(* Logix 5000 project; controller STAT 1756-L72 rev 20.12; software revision 20.04; part 7 of 34 *)
(* tags used below, declared in another part *)
   B11 : DINT[5];
   B15 : DINT[11];
   B3 : DINT[5];
   B9 : DINT[2];
   C5 : COUNTER[8];
   N17 : DINT[80];
   T10 : TIMER[30];
   T12 : TIMER[30];
   T4 : TIMER[30];
(* ECOTECH, continued *)

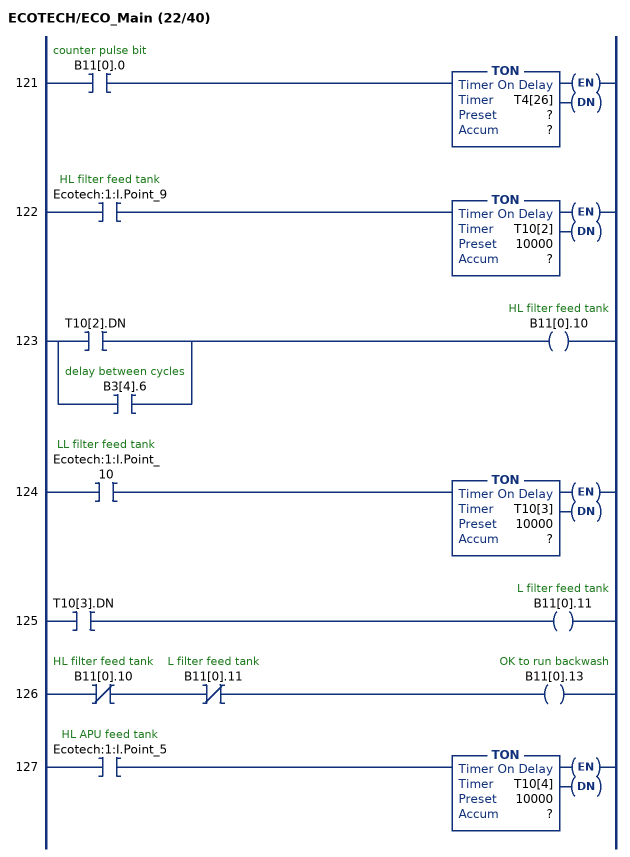
   [picture p70: ECOTECH/ECO_Main rungs 121-127]
   121: XIC(B11[0].0)TON(T4[26],?,?);
   122: XIC(Ecotech:1:I.Point_9)TON(T10[2],?,?);
   123: [XIC(T10[2].DN) ,XIC(B3[4].6) ]OTE(B11[0].10);
   124: XIC(Ecotech:1:I.Point_10)TON(T10[3],?,?);
   125: XIC(T10[3].DN)OTE(B11[0].11);
   126: XIO(B11[0].10)XIO(B11[0].11)OTE(B11[0].13);
   127: XIC(Ecotech:1:I.Point_5)TON(T10[4],?,?);
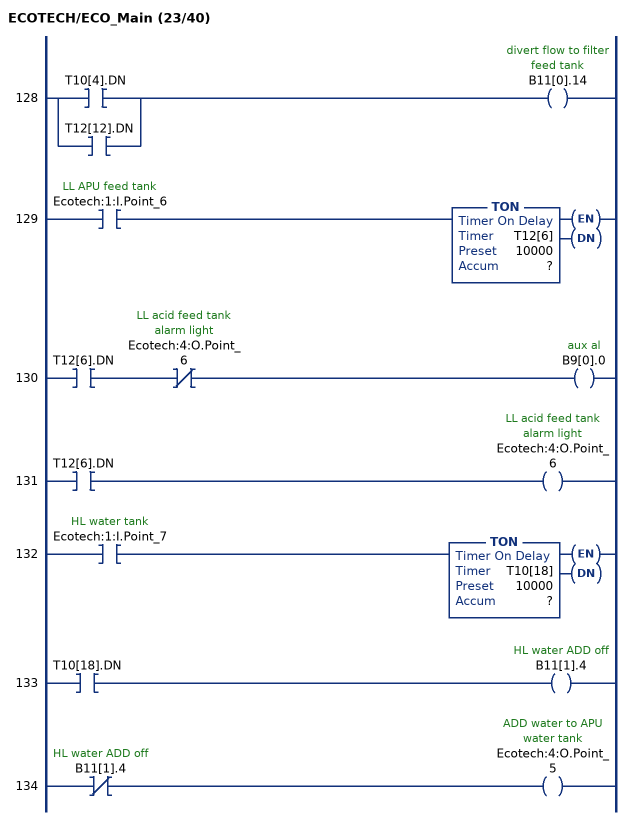
   128: [XIC(T10[4].DN) ,XIC(T12[12].DN) ]OTE(B11[0].14);
   129: XIC(Ecotech:1:I.Point_6)TON(T12[6],?,?);
   130: XIC(T12[6].DN)XIO(Ecotech:4:O.Point_6)OTE(B9[0].0);
   131: XIC(T12[6].DN)OTE(Ecotech:4:O.Point_6);
   132: XIC(Ecotech:1:I.Point_7)TON(T10[18],?,?);
   133: XIC(T10[18].DN)OTE(B11[1].4);
   134: XIO(B11[1].4)OTE(Ecotech:4:O.Point_5);
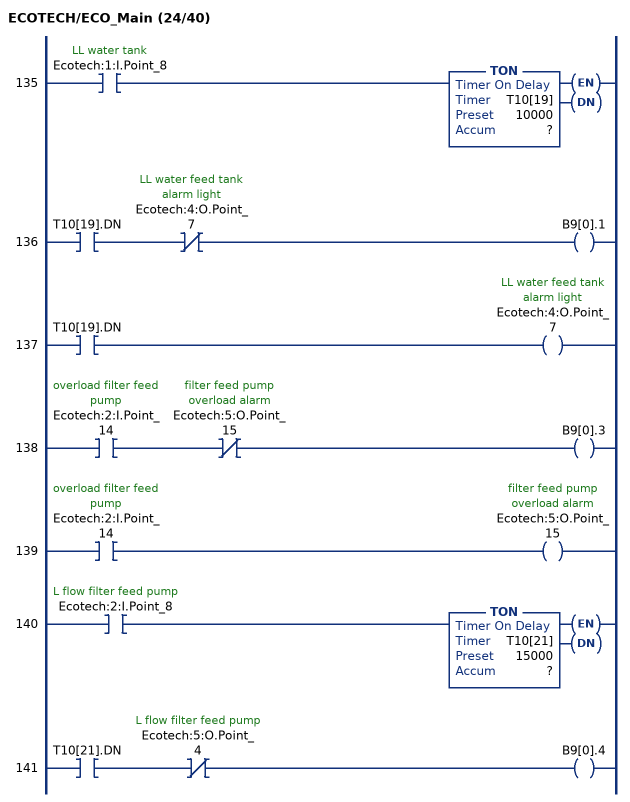
   135: XIC(Ecotech:1:I.Point_8)TON(T10[19],?,?);
   136: XIC(T10[19].DN)XIO(Ecotech:4:O.Point_7)OTE(B9[0].1);
   137: XIC(T10[19].DN)OTE(Ecotech:4:O.Point_7);
   138: XIC(Ecotech:2:I.Point_14)XIO(Ecotech:5:O.Point_15)OTE(B9[0].3);
   139: XIC(Ecotech:2:I.Point_14)OTE(Ecotech:5:O.Point_15);
   140: XIC(Ecotech:2:I.Point_8)TON(T10[21],?,?);
   141: XIC(T10[21].DN)XIO(Ecotech:5:O.Point_4)OTE(B9[0].4);
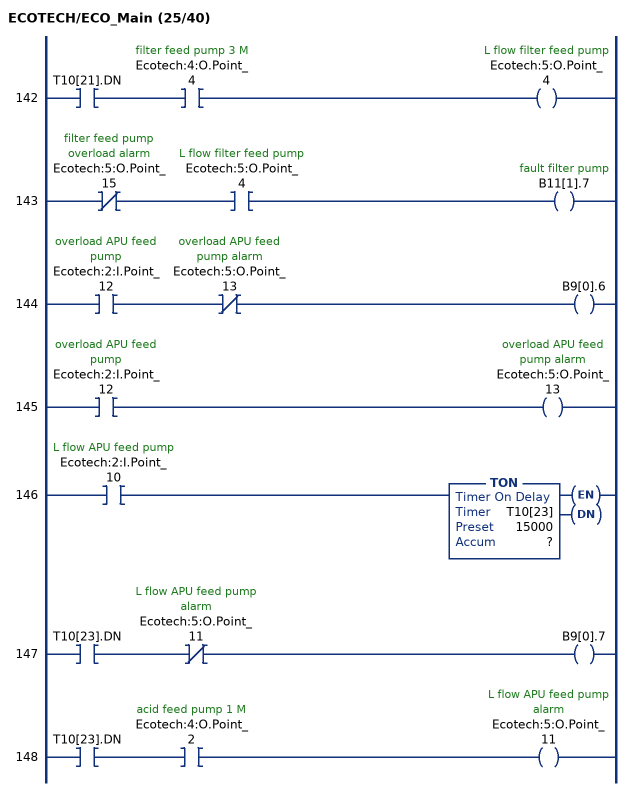
   142: XIC(T10[21].DN)XIC(Ecotech:4:O.Point_4)OTE(Ecotech:5:O.Point_4);
   143: XIO(Ecotech:5:O.Point_15)XIC(Ecotech:5:O.Point_4)OTE(B11[1].7);
   144: XIC(Ecotech:2:I.Point_12)XIO(Ecotech:5:O.Point_13)OTE(B9[0].6);
   145: XIC(Ecotech:2:I.Point_12)OTE(Ecotech:5:O.Point_13);
   146: XIC(Ecotech:2:I.Point_10)TON(T10[23],?,?);
   147: XIC(T10[23].DN)XIO(Ecotech:5:O.Point_11)OTE(B9[0].7);
   148: XIC(T10[23].DN)XIC(Ecotech:4:O.Point_2)OTE(Ecotech:5:O.Point_11);
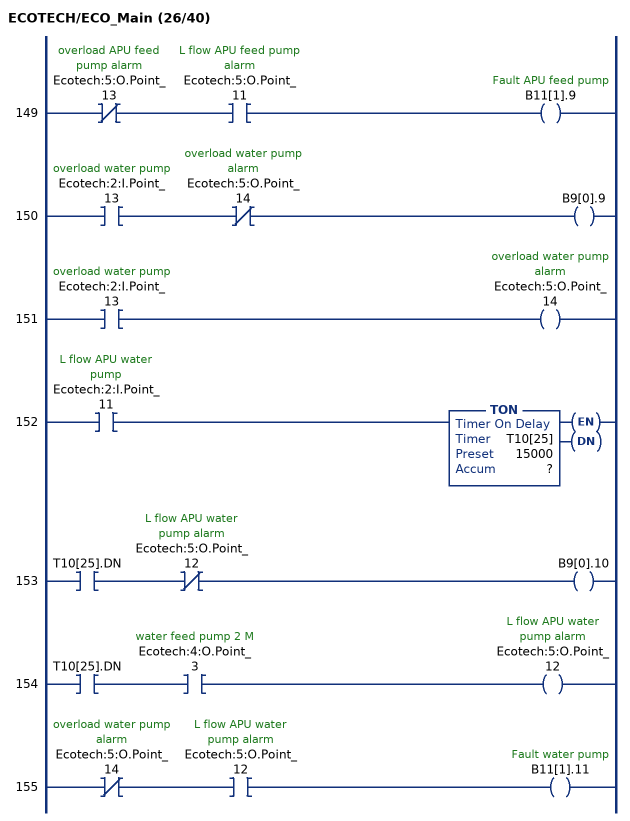
   149: XIO(Ecotech:5:O.Point_13)XIC(Ecotech:5:O.Point_11)OTE(B11[1].9);
   150: XIC(Ecotech:2:I.Point_13)XIO(Ecotech:5:O.Point_14)OTE(B9[0].9);
   151: XIC(Ecotech:2:I.Point_13)OTE(Ecotech:5:O.Point_14);
   152: XIC(Ecotech:2:I.Point_11)TON(T10[25],?,?);
   153: XIC(T10[25].DN)XIO(Ecotech:5:O.Point_12)OTE(B9[0].10);
   154: XIC(T10[25].DN)XIC(Ecotech:4:O.Point_3)OTE(Ecotech:5:O.Point_12);
   155: XIO(Ecotech:5:O.Point_14)XIC(Ecotech:5:O.Point_12)OTE(B11[1].11);
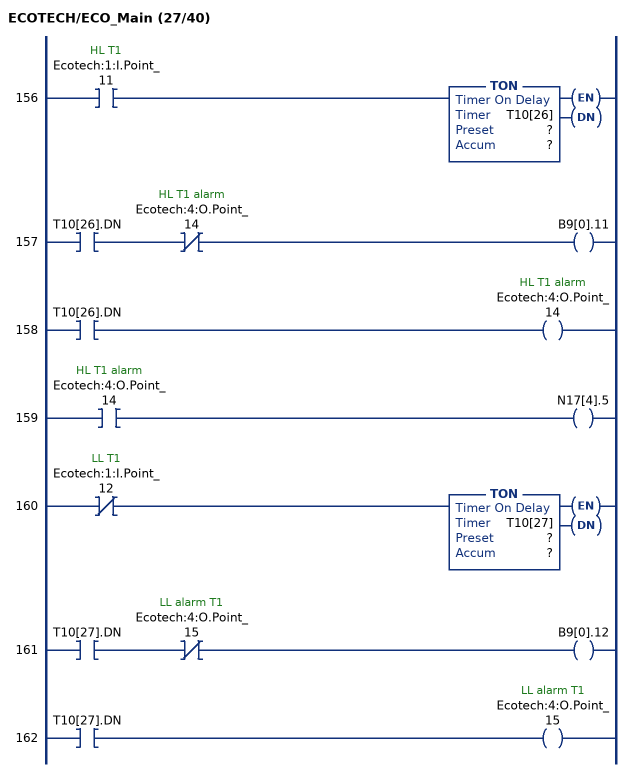
   156: XIC(Ecotech:1:I.Point_11)TON(T10[26],?,?);
   157: XIC(T10[26].DN)XIO(Ecotech:4:O.Point_14)OTE(B9[0].11);
   158: XIC(T10[26].DN)OTE(Ecotech:4:O.Point_14);
   159: XIC(Ecotech:4:O.Point_14)OTE(N17[4].5);
   160: XIO(Ecotech:1:I.Point_12)TON(T10[27],?,?);
   161: XIC(T10[27].DN)XIO(Ecotech:4:O.Point_15)OTE(B9[0].12);
   162: XIC(T10[27].DN)OTE(Ecotech:4:O.Point_15);
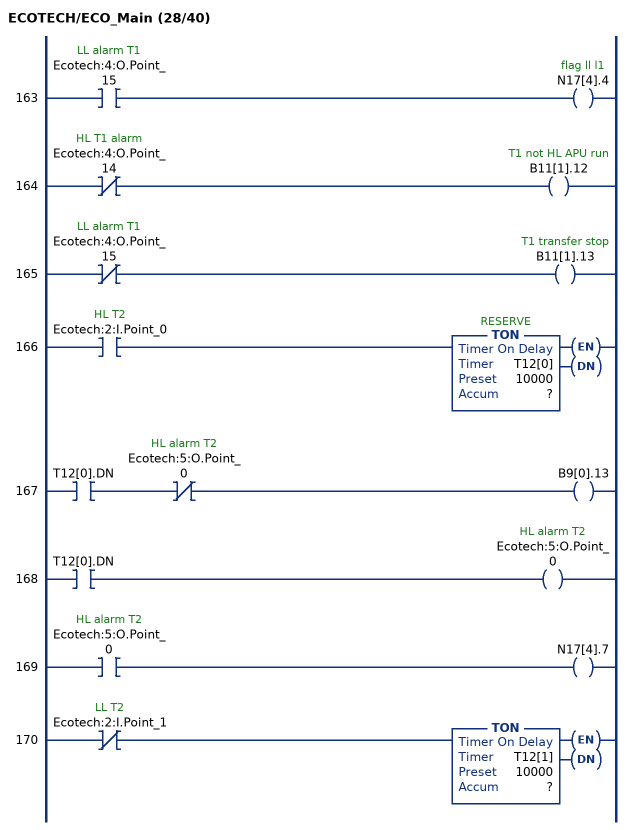
   163: XIC(Ecotech:4:O.Point_15)OTE(N17[4].4);
   164: XIO(Ecotech:4:O.Point_14)OTE(B11[1].12);
   165: XIO(Ecotech:4:O.Point_15)OTE(B11[1].13);
   166: XIC(Ecotech:2:I.Point_0)TON(T12[0],?,?);
   167: XIC(T12[0].DN)XIO(Ecotech:5:O.Point_0)OTE(B9[0].13);
   168: XIC(T12[0].DN)OTE(Ecotech:5:O.Point_0);
   169: XIC(Ecotech:5:O.Point_0)OTE(N17[4].7);
   170: XIO(Ecotech:2:I.Point_1)TON(T12[1],?,?);
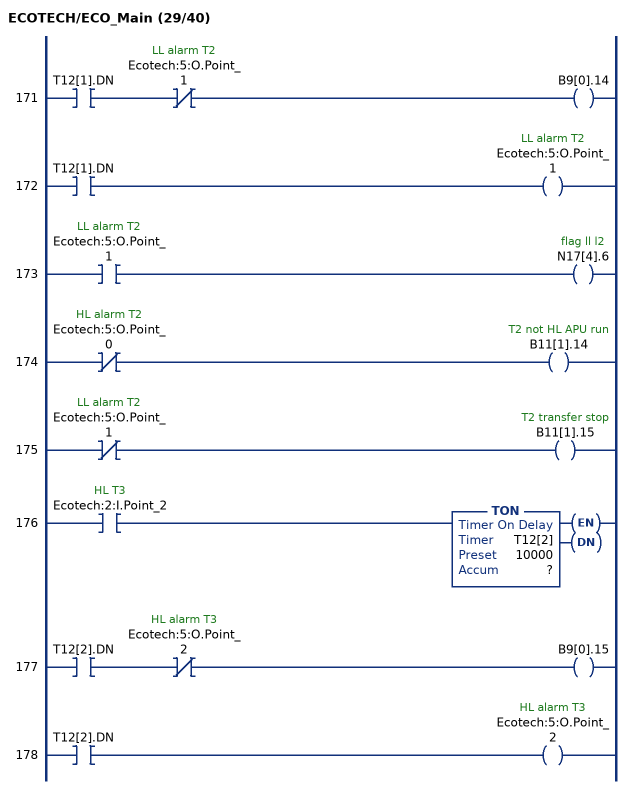
   171: XIC(T12[1].DN)XIO(Ecotech:5:O.Point_1)OTE(B9[0].14);
   172: XIC(T12[1].DN)OTE(Ecotech:5:O.Point_1);
   173: XIC(Ecotech:5:O.Point_1)OTE(N17[4].6);
   174: XIO(Ecotech:5:O.Point_0)OTE(B11[1].14);
   175: XIO(Ecotech:5:O.Point_1)OTE(B11[1].15);
   176: XIC(Ecotech:2:I.Point_2)TON(T12[2],?,?);
   177: XIC(T12[2].DN)XIO(Ecotech:5:O.Point_2)OTE(B9[0].15);
   178: XIC(T12[2].DN)OTE(Ecotech:5:O.Point_2);
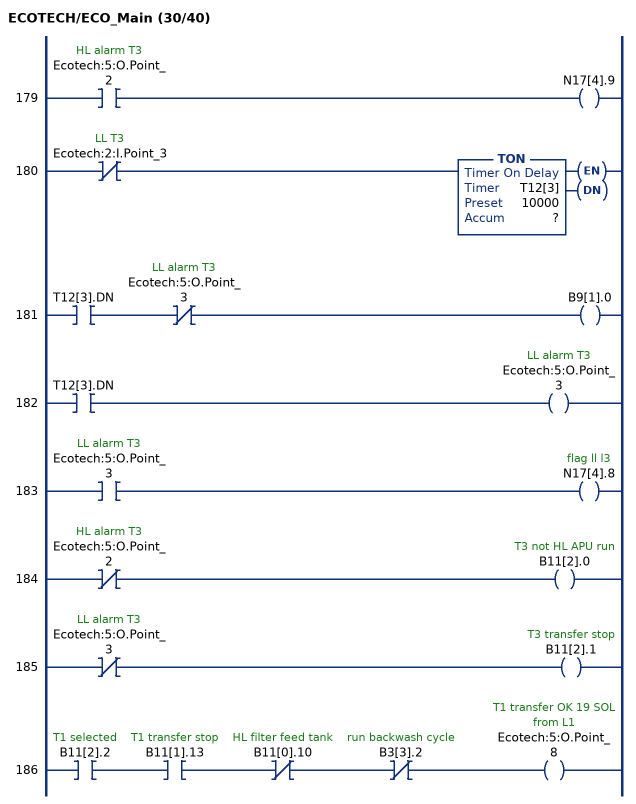
   179: XIC(Ecotech:5:O.Point_2)OTE(N17[4].9);
   180: XIO(Ecotech:2:I.Point_3)TON(T12[3],?,?);
   181: XIC(T12[3].DN)XIO(Ecotech:5:O.Point_3)OTE(B9[1].0);
   182: XIC(T12[3].DN)OTE(Ecotech:5:O.Point_3);
   183: XIC(Ecotech:5:O.Point_3)OTE(N17[4].8);
   184: XIO(Ecotech:5:O.Point_2)OTE(B11[2].0);
   185: XIO(Ecotech:5:O.Point_3)OTE(B11[2].1);
   186: XIC(B11[2].2)XIC(B11[1].13)XIO(B11[0].10)XIO(B3[3].2)OTE(Ecotech:5:O.Point_8);
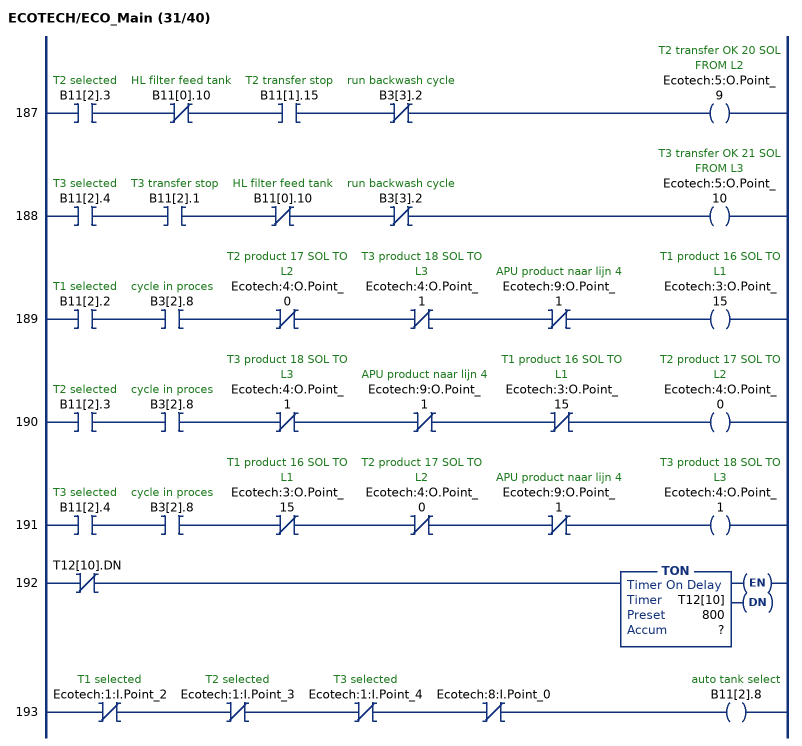
   187: XIC(B11[2].3)XIO(B11[0].10)XIC(B11[1].15)XIO(B3[3].2)OTE(Ecotech:5:O.Point_9);
   188: XIC(B11[2].4)XIC(B11[2].1)XIO(B11[0].10)XIO(B3[3].2)OTE(Ecotech:5:O.Point_10);
   189: XIC(B11[2].2)XIC(B3[2].8)XIO(Ecotech:4:O.Point_0)XIO(Ecotech:4:O.Point_1)XIO(Ecotech:9:O.Point_1)OTE(Ecotech:3:O.Point_15);
   190: XIC(B11[2].3)XIC(B3[2].8)XIO(Ecotech:4:O.Point_1)XIO(Ecotech:9:O.Point_1)XIO(Ecotech:3:O.Point_15)OTE(Ecotech:4:O.Point_0);
   191: XIC(B11[2].4)XIC(B3[2].8)XIO(Ecotech:3:O.Point_15)XIO(Ecotech:4:O.Point_0)XIO(Ecotech:9:O.Point_1)OTE(Ecotech:4:O.Point_1);
   192: XIO(T12[10].DN)TON(T12[10],?,?);
   193: XIO(Ecotech:1:I.Point_2)XIO(Ecotech:1:I.Point_3)XIO(Ecotech:1:I.Point_4)XIO(Ecotech:8:I.Point_0)OTE(B11[2].8);
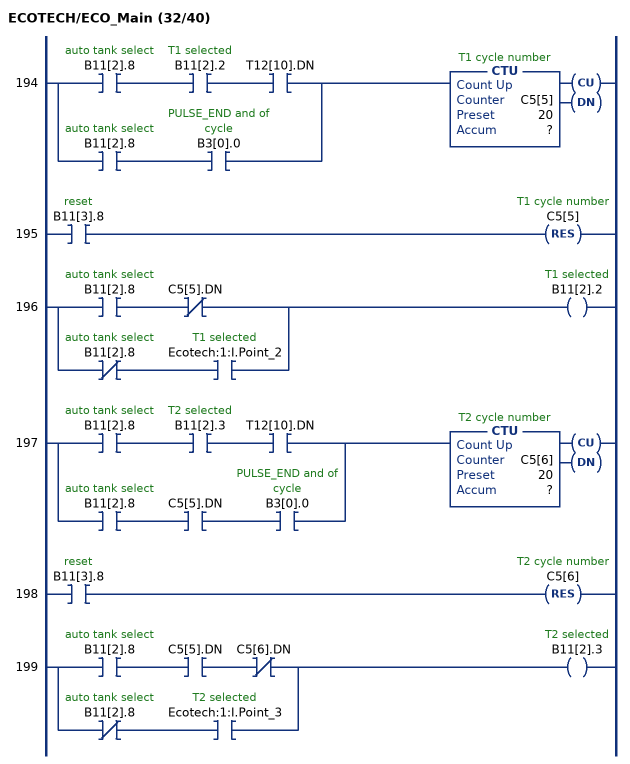
   194: [XIC(B11[2].8) XIC(B11[2].2) XIC(T12[10].DN) ,XIC(B11[2].8) XIC(B3[0].0) ]CTU(C5[5],?,?);
   195: XIC(B11[3].8)RES(C5[5]);
   196: [XIC(B11[2].8) XIO(C5[5].DN) ,XIO(B11[2].8) XIC(Ecotech:1:I.Point_2) ]OTE(B11[2].2);
   197: [XIC(B11[2].8) XIC(B11[2].3) XIC(T12[10].DN) ,XIC(B11[2].8) XIC(C5[5].DN) XIC(B3[0].0) ]CTU(C5[6],?,?);
   198: XIC(B11[3].8)RES(C5[6]);
   199: [XIC(B11[2].8) XIC(C5[5].DN) XIO(C5[6].DN) ,XIO(B11[2].8) XIC(Ecotech:1:I.Point_3) ]OTE(B11[2].3);
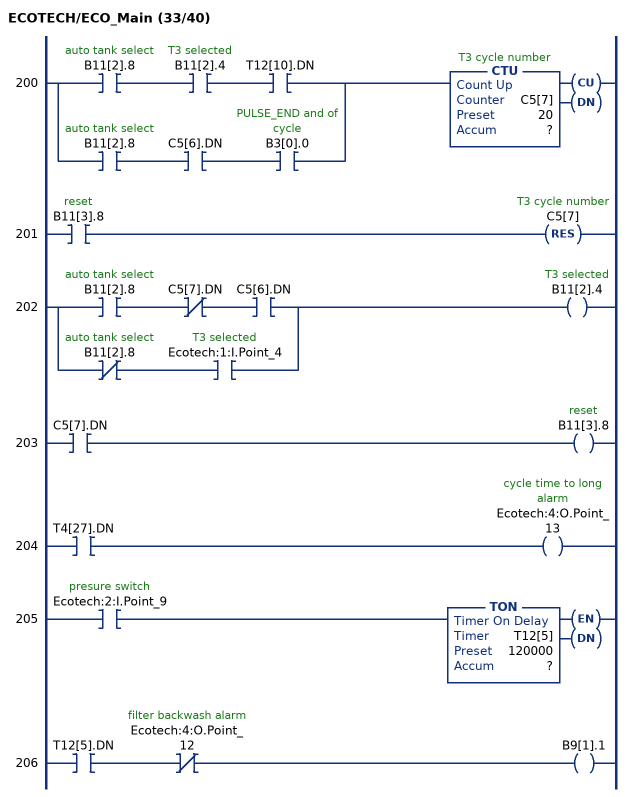
   200: [XIC(B11[2].8) XIC(B11[2].4) XIC(T12[10].DN) ,XIC(B11[2].8) XIC(C5[6].DN) XIC(B3[0].0) ]CTU(C5[7],?,?);
   201: XIC(B11[3].8)RES(C5[7]);
   202: [XIC(B11[2].8) XIO(C5[7].DN) XIC(C5[6].DN) ,XIO(B11[2].8) XIC(Ecotech:1:I.Point_4) ]OTE(B11[2].4);
   203: XIC(C5[7].DN)OTE(B11[3].8);
   204: XIC(T4[27].DN)OTE(Ecotech:4:O.Point_13);
   205: XIC(Ecotech:2:I.Point_9)TON(T12[5],?,?);
   206: XIC(T12[5].DN)XIO(Ecotech:4:O.Point_12)OTE(B9[1].1);
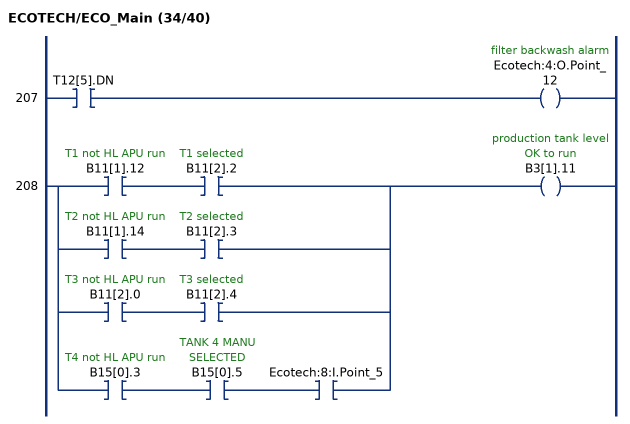
   207: XIC(T12[5].DN)OTE(Ecotech:4:O.Point_12);
   208: [XIC(B11[1].12) XIC(B11[2].2) ,XIC(B11[1].14) XIC(B11[2].3) ,XIC(B11[2].0) XIC(B11[2].4) ,XIC(B15[0].3) XIC(B15[0].5) XIC(Ecotech:8:I.Point_5) ]OTE(B3[1].11);
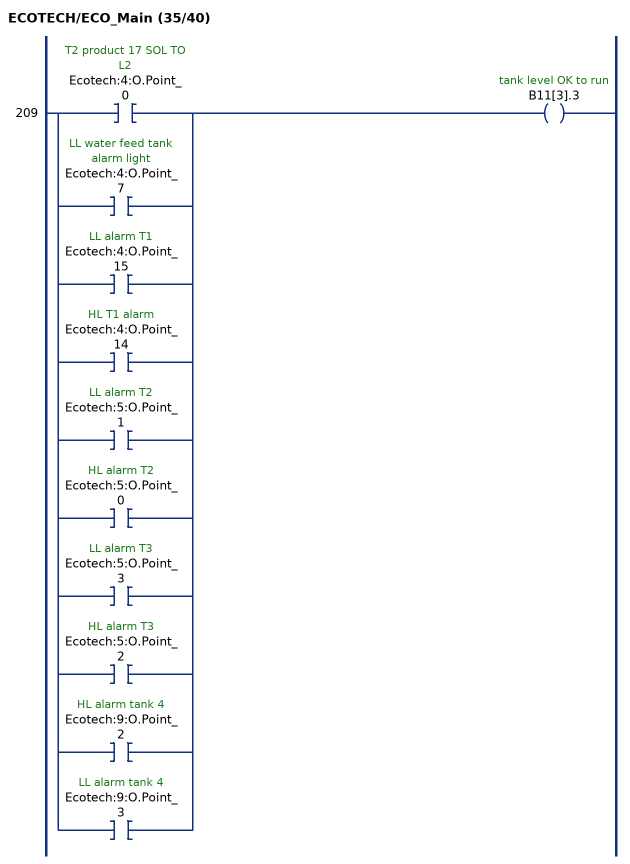
   209: [XIC(Ecotech:4:O.Point_0) ,XIC(Ecotech:4:O.Point_7) ,XIC(Ecotech:4:O.Point_15) ,XIC(Ecotech:4:O.Point_14) ,XIC(Ecotech:5:O.Point_1) ,XIC(Ecotech:5:O.Point_0) ,XIC(Ecotech:5:O.Point_3) ,XIC(Ecotech:5:O.Point_2) ,XIC(Ecotech:9:O.Point_2) ,XIC(Ecotech:9:O.Point_3) ]OTE(B11[3].3);
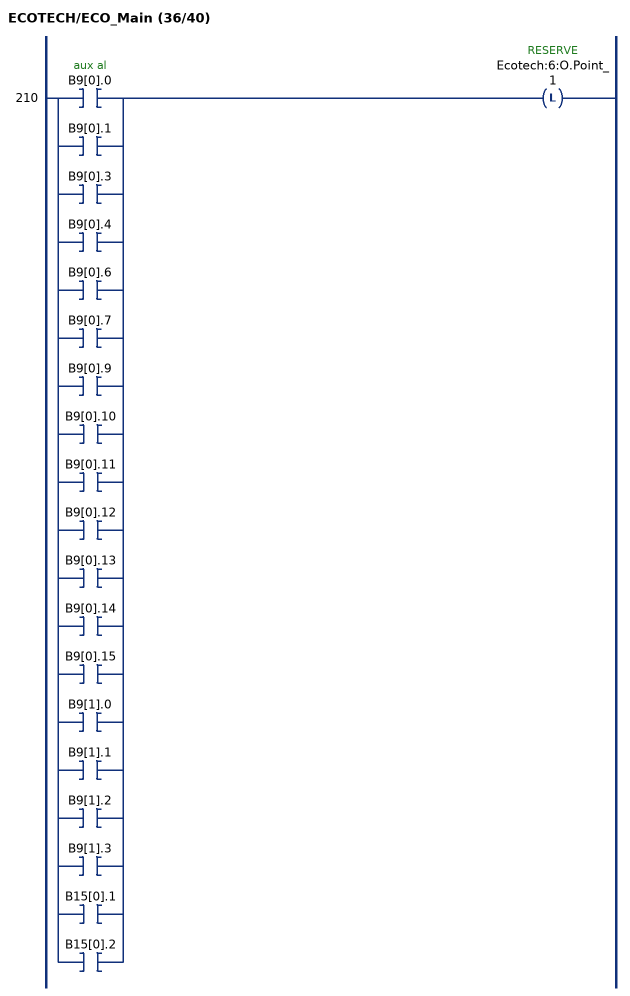
   210: [XIC(B9[0].0) ,XIC(B9[0].1) ,XIC(B9[0].3) ,XIC(B9[0].4) ,XIC(B9[0].6) ,XIC(B9[0].7) ,XIC(B9[0].9) ,XIC(B9[0].10) ,XIC(B9[0].11) ,XIC(B9[0].12) ,XIC(B9[0].13) ,XIC(B9[0].14) ,XIC(B9[0].15) ,XIC(B9[1].0) ,XIC(B9[1].1) ,XIC(B9[1].2) ,XIC(B9[1].3) ,XIC(B15[0].1) ,XIC(B15[0].2) ]OTL(Ecotech:6:O.Point_1);
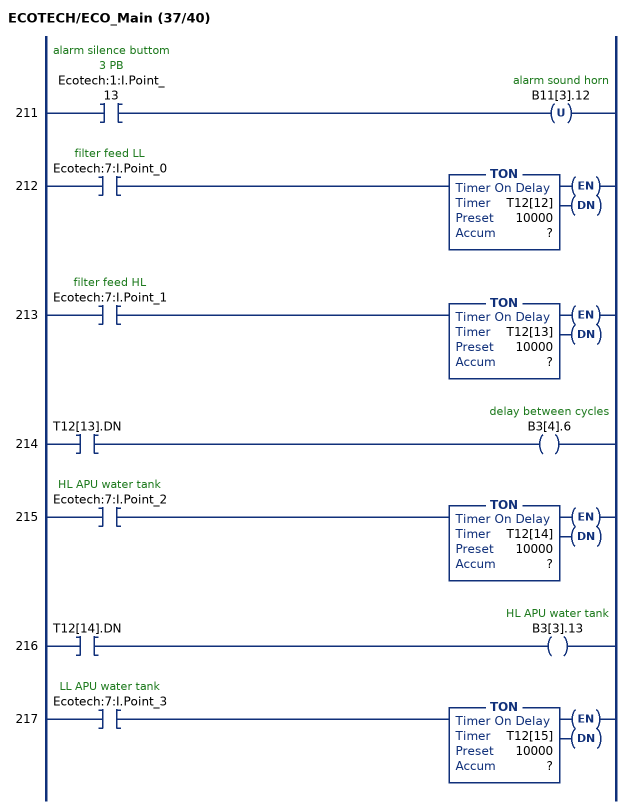
   211: XIC(Ecotech:1:I.Point_13)OTU(B11[3].12);
   212: XIC(Ecotech:7:I.Point_0)TON(T12[12],?,?);
   213: XIC(Ecotech:7:I.Point_1)TON(T12[13],?,?);
   214: XIC(T12[13].DN)OTE(B3[4].6);
   215: XIC(Ecotech:7:I.Point_2)TON(T12[14],?,?);
   216: XIC(T12[14].DN)OTE(B3[3].13);
   217: XIC(Ecotech:7:I.Point_3)TON(T12[15],?,?);
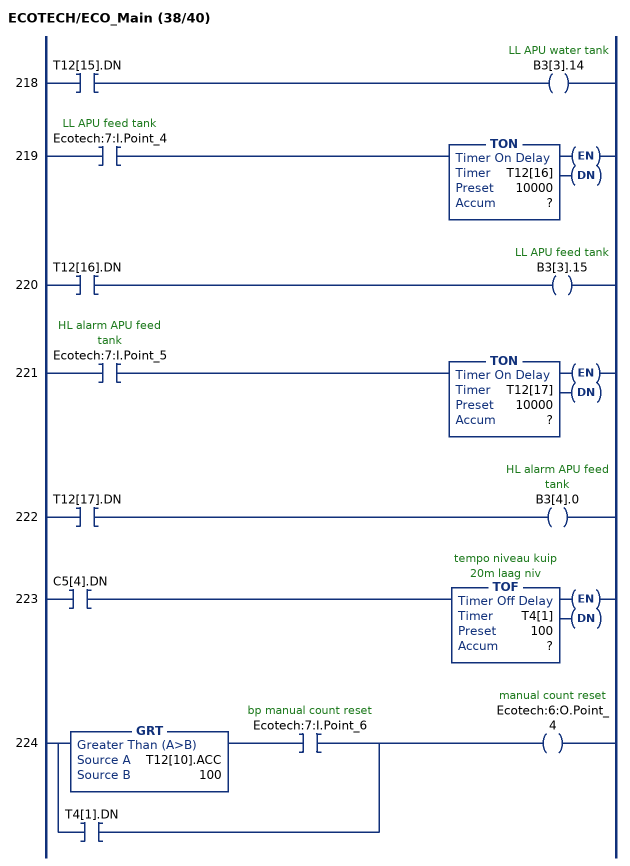
   218: XIC(T12[15].DN)OTE(B3[3].14);
   219: XIC(Ecotech:7:I.Point_4)TON(T12[16],?,?);
   220: XIC(T12[16].DN)OTE(B3[3].15);
   221: XIC(Ecotech:7:I.Point_5)TON(T12[17],?,?);
   222: XIC(T12[17].DN)OTE(B3[4].0);
   223: XIC(C5[4].DN)TOF(T4[1],?,?);
   224: [GRT(T12[10].ACC,100) XIC(Ecotech:7:I.Point_6) ,XIC(T4[1].DN) ]OTE(Ecotech:6:O.Point_4);
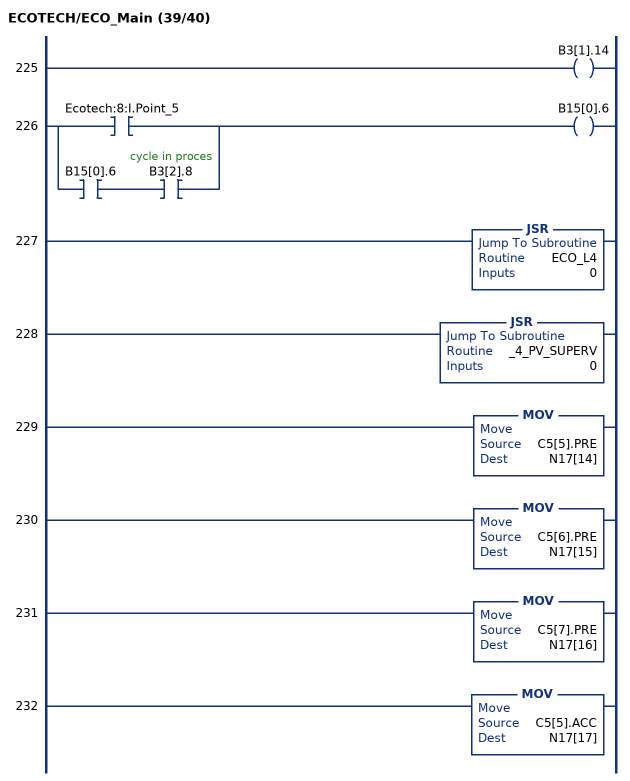
   225: OTE(B3[1].14);
   226: [XIC(Ecotech:8:I.Point_5) ,XIC(B15[0].6) XIC(B3[2].8) ]OTE(B15[0].6);
   227: JSR(ECO_L4,0);
   228: JSR(_4_PV_SUPERV,0);
   229: MOV(C5[5].PRE,N17[14]);
   230: MOV(C5[6].PRE,N17[15]);
   231: MOV(C5[7].PRE,N17[16]);
   232: MOV(C5[5].ACC,N17[17]);
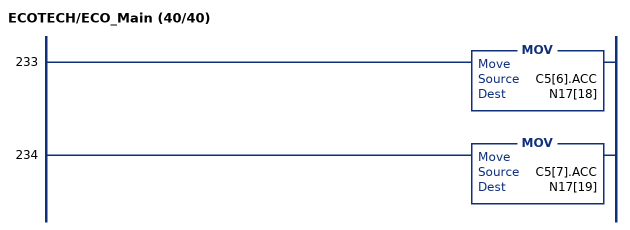
   233: MOV(C5[6].ACC,N17[18]);
   234: MOV(C5[7].ACC,N17[19]);
END_ROUTINE
END_PROGRAM
